TYPE (* A Structure with 16 BOOLS *)
  (* Version 1.0, 2024-02-21, Franz Höpfinger, HR Agrartechnik GmbH *)
  ST32B : STRUCT
    B_00 : BOOL; (* BIT 00 *)
    B_01 : BOOL; (* BIT 01 *)
    B_02 : BOOL; (* BIT 02 *)
    B_03 : BOOL; (* BIT 03 *)
    B_04 : BOOL; (* BIT 04 *)
    B_05 : BOOL; (* BIT 05 *)
    B_06 : BOOL; (* BIT 06 *)
    B_07 : BOOL; (* BIT 07 *)
    B_08 : BOOL; (* BIT 08 *)
    B_09 : BOOL; (* BIT 09 *)
    B_10 : BOOL; (* BIT 10 *)
    B_11 : BOOL; (* BIT 11 *)
    B_12 : BOOL; (* BIT 12 *)
    B_13 : BOOL; (* BIT 13 *)
    B_14 : BOOL; (* BIT 14 *)
    B_15 : BOOL; (* BIT 15 *)
    B_16 : BOOL; (* BIT 16 *)
    B_17 : BOOL; (* BIT 17 *)
    B_18 : BOOL; (* BIT 18 *)
    B_19 : BOOL; (* BIT 19 *)
    B_20 : BOOL; (* BIT 20 *)
    B_21 : BOOL; (* BIT 21 *)
    B_22 : BOOL; (* BIT 22 *)
    B_23 : BOOL; (* BIT 23 *)
    B_24 : BOOL; (* BIT 24 *)
    B_25 : BOOL; (* BIT 25 *)
    B_26 : BOOL; (* BIT 26 *)
    B_27 : BOOL; (* BIT 27 *)
    B_28 : BOOL; (* BIT 28 *)
    B_29 : BOOL; (* BIT 29 *)
    B_30 : BOOL; (* BIT 30 *)
    B_31 : BOOL; (* BIT 31 *)
  END_STRUCT;
END_TYPE
